// TIA Portal V17 export
// export: Created 2023-05-31T13:25:23.2864469Z, ExportSetting WithDefaults, DisplayName Totally Integrated Automation Portal, DisplayVersion V17, DisplayName TIA Portal Openness, DisplayVersion V17, DisplayName TIA Portal Version Control Interface, DisplayVersion V17, DisplayName STEP 7 Professional, DisplayVersion V17, DisplayName STEP 7 Safety, DisplayVersion V17, DisplayName WinCC Advanced, DisplayVersion V17
DATA_BLOCK "FB_Unit_EDUKIT_PA_Control_DB"   // DB2
VERSION : 0.1
// stored: AutoNumber true, DBAccessibleFromOPCUA true, InstanceOfName FB_Unit_EDUKIT_PA_Control, InstanceOfType FB
"FB_Unit_EDUKIT_PA_Control"
   // VAR_INPUT
   //    Ainput_0 : Int;
   //    Ainput_1 : Int;
   //    Ainput_2 : Int;
   // END_VAR
   // VAR_OUTPUT
   //    output_startMotor : Bool;
   //    "output_motorPower [%]" : Real;
   //    output_valve : Bool;
   // END_VAR
   // VAR
   //    startMotor : Bool;
   //    "motorPower [%]" : Real;
   //    valve : Bool;
   //    "Flow [l/h]" : Real;
   //    "pressure [mbar]" : Real;
   //    "pressure [psi]" : Real;
   //    "level [l]" : Real;
   //    "step" : Array[0..20] of Bool;
   // END_VAR
BEGIN
END_DATA_BLOCK
